{attribute addProperty BoxType "EJ6224-0000-0016"}
{attribute addProperty Id "DeviceState_InputsDeviceState_Inputs_BDC6BEC3324"}
{attribute addProperty CRC "3630215907"}
{attribute addProperty SizeInBites "32"}
{attribute addProperty SizeInBytes "4"}
TYPE Module_2_DeviceState_Inputs_D860B2E3 :
STRUCT
	{attribute addProperty Name "DeviceState_Inputs"}
	DeviceState_Inputs  : DeviceState_Inputs_BDC6BEC3;
END_STRUCT
END_TYPE

(* stored: Version 1.2.0.0, ProductVersion 3.1.4024.9
   DUT Module_2_DeviceState_Inputs_D860B2E3: Id {7f327a3a-a6d3-44f2-a63a-3b1177dca762} *)
